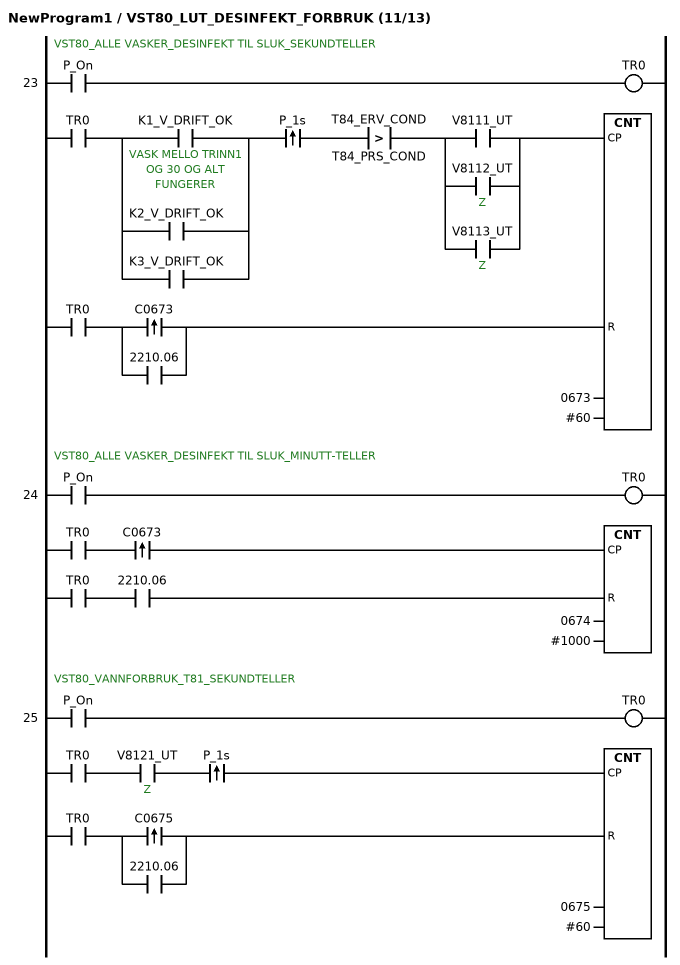
; [picture p24: NewProgram1 / VST80_LUT_DESINFEKT_FORBRUK, rungs 23-25]
; rung 23: VST80_ALLE VASKER_DESINFEKT TIL SLUK_SEKUNDTELLER
LD P_On
OUT TR0
LD K1_V_DRIFT_OK  ; VASK MELLO TRINN1 OG 30 OG ALT FUNGERER
OR K2_V_DRIFT_OK
OR K3_V_DRIFT_OK
ANDLD
@AND P_1s
AND>(320) T84_ERV_COND T84_PRS_COND
LD V8111_UT
OR V8112_UT  ; Z
OR V8113_UT  ; Z
ANDLD
LD TR0
@LD C0673
OR 2210.06
ANDLD
CNT 0673 #60
; rung 24: VST80_ALLE VASKER_DESINFEKT TIL SLUK_MINUTT-TELLER
LD P_On
OUT TR0
@AND C0673
LD TR0
AND 2210.06
CNT 0674 #1000
; rung 25: VST80_VANNFORBRUK_T81_SEKUNDTELLER
LD P_On
OUT TR0
AND V8121_UT  ; Z
@AND P_1s
LD TR0
@LD C0675
OR 2210.06
ANDLD
CNT 0675 #60

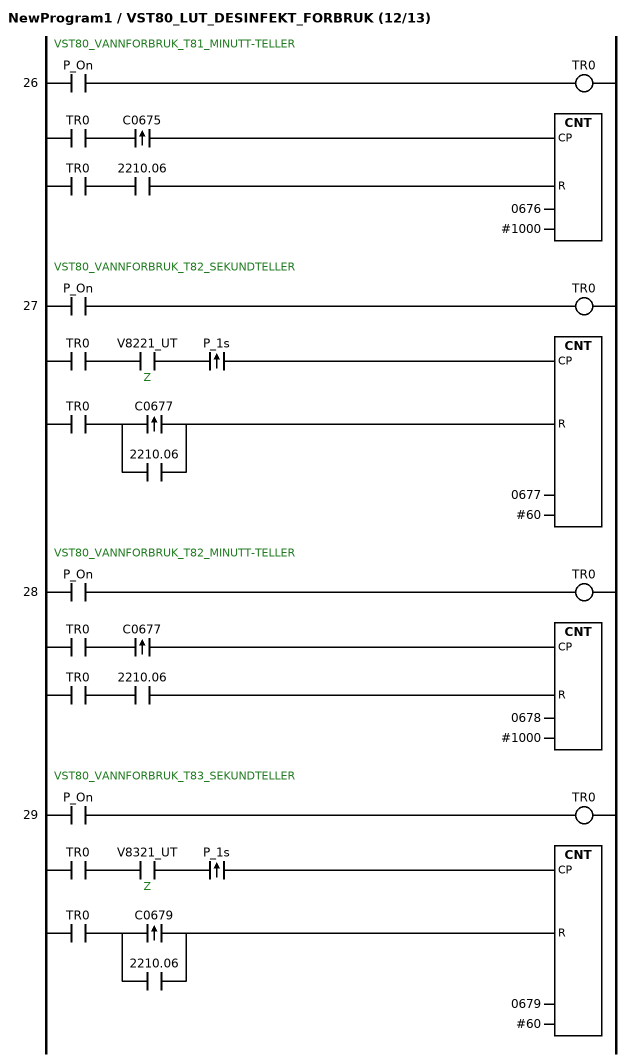
; rung 26: VST80_VANNFORBRUK_T81_MINUTT-TELLER
LD P_On
OUT TR0
@AND C0675
LD TR0
AND 2210.06
CNT 0676 #1000
; rung 27: VST80_VANNFORBRUK_T82_SEKUNDTELLER
LD P_On
OUT TR0
AND V8221_UT  ; Z
@AND P_1s
LD TR0
@LD C0677
OR 2210.06
ANDLD
CNT 0677 #60
; rung 28: VST80_VANNFORBRUK_T82_MINUTT-TELLER
LD P_On
OUT TR0
@AND C0677
LD TR0
AND 2210.06
CNT 0678 #1000
; rung 29: VST80_VANNFORBRUK_T83_SEKUNDTELLER
LD P_On
OUT TR0
AND V8321_UT  ; Z
@AND P_1s
LD TR0
@LD C0679
OR 2210.06
ANDLD
CNT 0679 #60

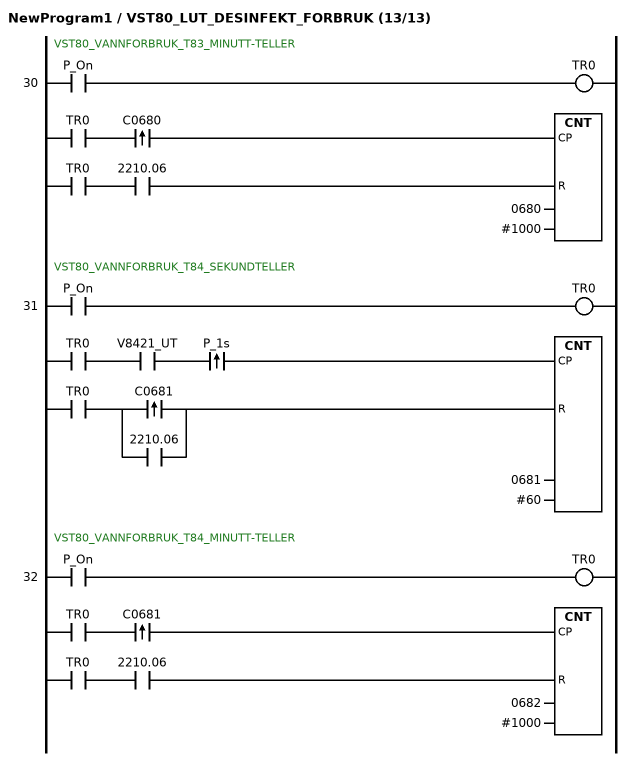
; rung 30: VST80_VANNFORBRUK_T83_MINUTT-TELLER
LD P_On
OUT TR0
@AND C0680
LD TR0
AND 2210.06
CNT 0680 #1000
; rung 31: VST80_VANNFORBRUK_T84_SEKUNDTELLER
LD P_On
OUT TR0
AND V8421_UT
@AND P_1s
LD TR0
@LD C0681
OR 2210.06
ANDLD
CNT 0681 #60
; rung 32: VST80_VANNFORBRUK_T84_MINUTT-TELLER
LD P_On
OUT TR0
@AND C0681
LD TR0
AND 2210.06
CNT 0682 #1000
; rung 33: Ingen_kommentar_funnet

### Section T81_NIVÅ

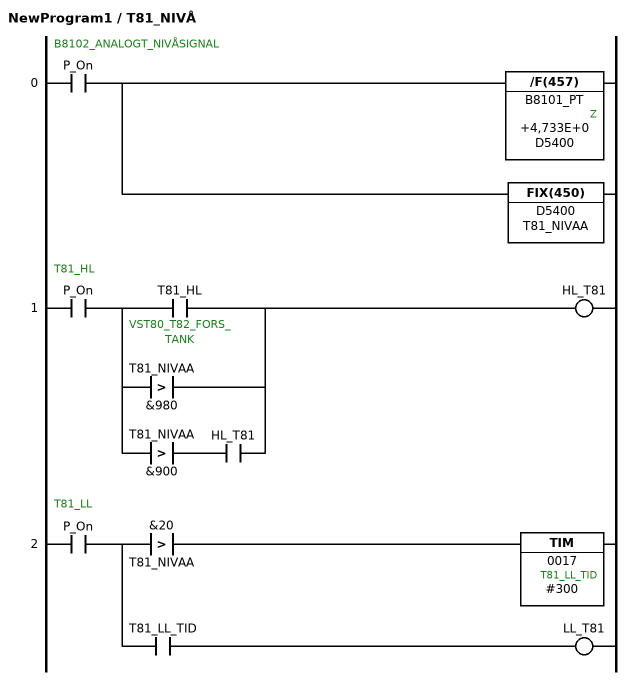
; rung 0: B8102_ANALOGT_NIVÅSIGNAL
LD P_On
/F(457) B8101_PT +4,733E+0 D5400  ; Z
FIX(450) D5400 T81_NIVAA
; rung 1: T81_HL
LD P_On
LD T81_HL  ; VST80_T82_FORS_TANK
OR>(320) T81_NIVAA &980
LD>(320) T81_NIVAA &900
AND HL_T81
ORLD
ANDLD
OUT HL_T81
; rung 2: T81_LL
LD P_On
OUT TR0
AND>(320) &20 T81_NIVAA
TIM 0017 #300  ; T81_LL_TID
LD TR0
AND T81_LL_TID
OUT LL_T81
; rung 3: Ingen_kommentar_funnet

### Section T81_FUNKSJONER_OBJEKTER
; Dette programmet styrer kommandoene til vaskestasjonen.

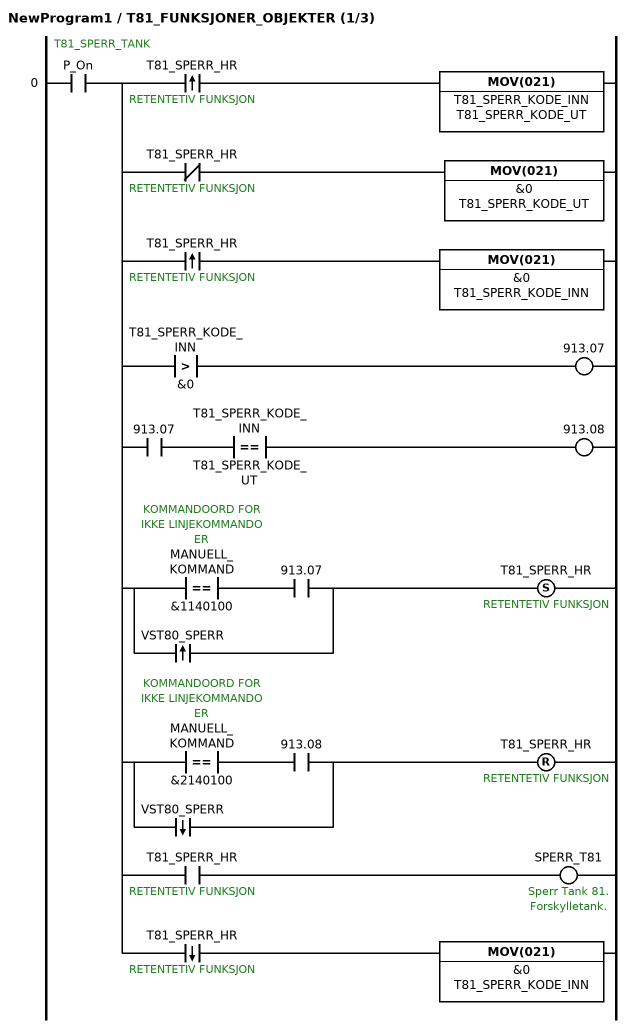
; rung 0: T81_SPERR_TANK
LD P_On
OUT TR0
@AND T81_SPERR_HR  ; RETENTETIV FUNKSJON
MOV(021) T81_SPERR_KODE_INN T81_SPERR_KODE_UT
LD TR0
ANDNOT T81_SPERR_HR  ; RETENTETIV FUNKSJON
MOV(021) &0 T81_SPERR_KODE_UT
LD TR0
@AND T81_SPERR_HR  ; RETENTETIV FUNKSJON
MOV(021) &0 T81_SPERR_KODE_INN
LD TR0
AND>(320) T81_SPERR_KODE_INN &0
OUT 913.07
LD TR0
AND 913.07
AND=(300) T81_SPERR_KODE_INN T81_SPERR_KODE_UT
OUT 913.08
LD TR0
LD=L(301) MANUELL_KOMMAND &1140100  ; KOMMANDOORD FOR IKKE LINJEKOMMANDOER
AND 913.07
@OR VST80_SPERR
ANDLD
SET T81_SPERR_HR  ; RETENTETIV FUNKSJON
LD TR0
LD=L(301) MANUELL_KOMMAND &2140100  ; KOMMANDOORD FOR IKKE LINJEKOMMANDOER
AND 913.08
%OR VST80_SPERR
ANDLD
RSET T81_SPERR_HR  ; RETENTETIV FUNKSJON
LD TR0
AND T81_SPERR_HR  ; RETENTETIV FUNKSJON
OUT SPERR_T81  ; Sperr Tank 81. Forskylletank.
LD TR0
%AND T81_SPERR_HR  ; RETENTETIV FUNKSJON
MOV(021) &0 T81_SPERR_KODE_INN

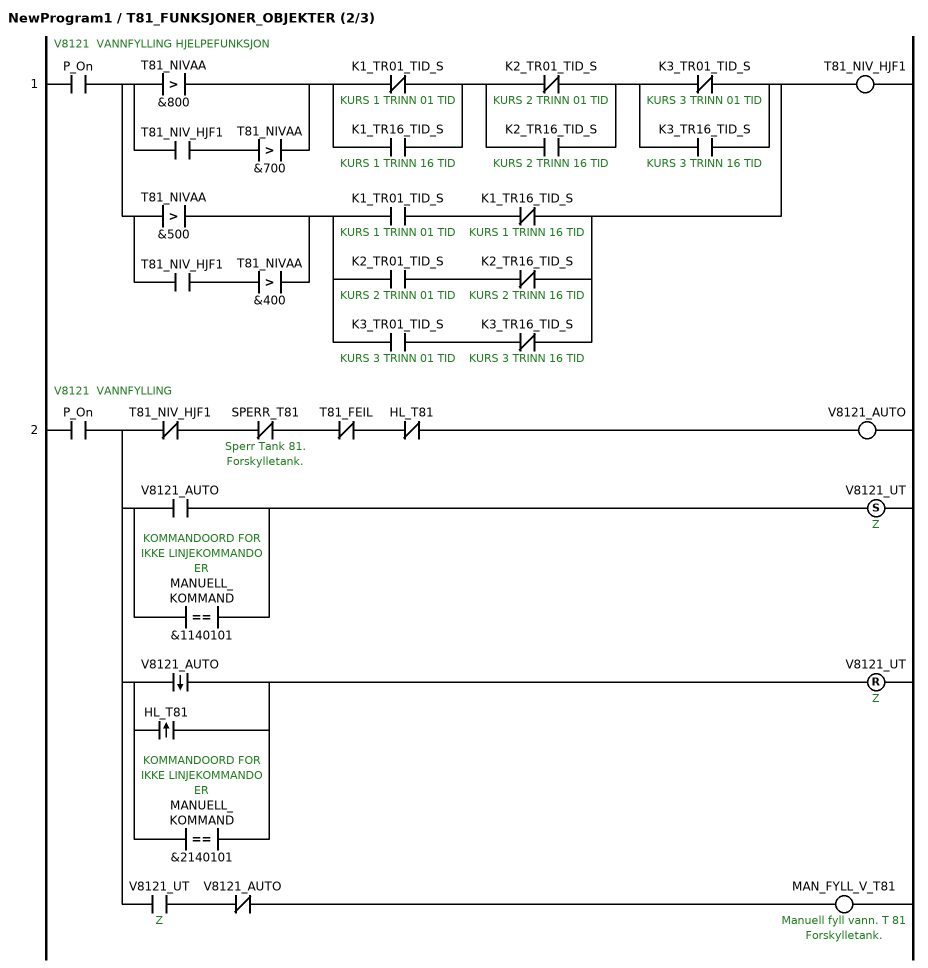
; rung 1: V8121  VANNFYLLING HJELPEFUNKSJON
LD P_On
LD>(320) T81_NIVAA &800
LD T81_NIV_HJF1
AND>(320) T81_NIVAA &700
ORLD
LDNOT K1_TR01_TID_S  ; KURS 1 TRINN 01 TID
OR K1_TR16_TID_S  ; KURS 1 TRINN 16 TID
ANDLD
LDNOT K2_TR01_TID_S  ; KURS 2 TRINN 01 TID
OR K2_TR16_TID_S  ; KURS 2 TRINN 16 TID
ANDLD
LDNOT K3_TR01_TID_S  ; KURS 3 TRINN 01 TID
OR K3_TR16_TID_S  ; KURS 3 TRINN 16 TID
ANDLD
LD>(320) T81_NIVAA &500
LD T81_NIV_HJF1
AND>(320) T81_NIVAA &400
ORLD
LD K1_TR01_TID_S  ; KURS 1 TRINN 01 TID
ANDNOT K1_TR16_TID_S  ; KURS 1 TRINN 16 TID
LD K2_TR01_TID_S  ; KURS 2 TRINN 01 TID
ANDNOT K2_TR16_TID_S  ; KURS 2 TRINN 16 TID
ORLD
LD K3_TR01_TID_S  ; KURS 3 TRINN 01 TID
ANDNOT K3_TR16_TID_S  ; KURS 3 TRINN 16 TID
ORLD
ANDLD
ORLD
ANDLD
OUT T81_NIV_HJF1
; rung 2: V8121  VANNFYLLING
LD P_On
OUT TR0
ANDNOT T81_NIV_HJF1
ANDNOT SPERR_T81  ; Sperr Tank 81. Forskylletank.
ANDNOT T81_FEIL
ANDNOT HL_T81
OUT V8121_AUTO
LD TR0
LD V8121_AUTO
OR=L(301) MANUELL_KOMMAND &1140101  ; KOMMANDOORD FOR IKKE LINJEKOMMANDOER
ANDLD
SET V8121_UT  ; Z
LD TR0
%LD V8121_AUTO
@OR HL_T81
OR=L(301) MANUELL_KOMMAND &2140101  ; KOMMANDOORD FOR IKKE LINJEKOMMANDOER
ANDLD
RSET V8121_UT  ; Z
LD TR0
AND V8121_UT  ; Z
ANDNOT V8121_AUTO
OUT MAN_FYLL_V_T81  ; Manuell fyll vann. T 81 Forskylletank.

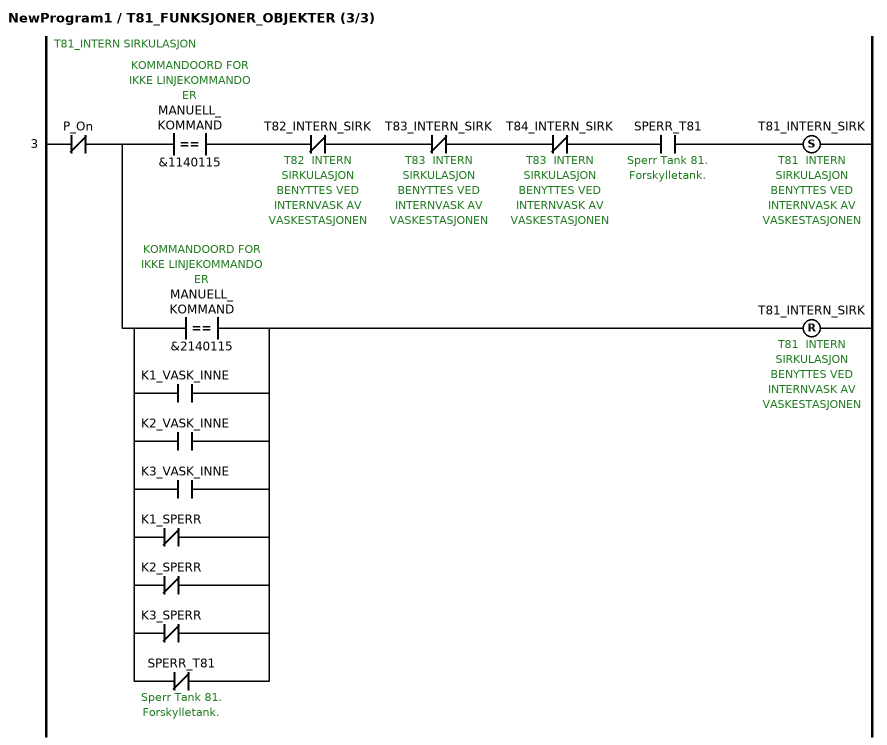
; rung 3: T81_INTERN SIRKULASJON
LDNOT P_On
OUT TR0
AND=L(301) MANUELL_KOMMAND &1140115  ; KOMMANDOORD FOR IKKE LINJEKOMMANDOER
ANDNOT T82_INTERN_SIRK  ; T82  INTERN SIRKULASJON BENYTTES VED INTERNVASK AV VASKESTASJONEN
ANDNOT T83_INTERN_SIRK  ; T83  INTERN SIRKULASJON BENYTTES VED INTERNVASK AV VASKESTASJONEN
ANDNOT T84_INTERN_SIRK  ; T83  INTERN SIRKULASJON BENYTTES VED INTERNVASK AV VASKESTASJONEN
AND SPERR_T81  ; Sperr Tank 81. Forskylletank.
SET T81_INTERN_SIRK  ; T81  INTERN SIRKULASJON BENYTTES VED INTERNVASK AV VASKESTASJONEN
LD TR0
LD=L(301) MANUELL_KOMMAND &2140115  ; KOMMANDOORD FOR IKKE LINJEKOMMANDOER
OR K1_VASK_INNE
OR K2_VASK_INNE
OR K3_VASK_INNE
ORNOT K1_SPERR
ORNOT K2_SPERR
ORNOT K3_SPERR
ORNOT SPERR_T81  ; Sperr Tank 81. Forskylletank.
ANDLD
RSET T81_INTERN_SIRK  ; T81  INTERN SIRKULASJON BENYTTES VED INTERNVASK AV VASKESTASJONEN
; rung 4: Ingen_kommentar_funnet

### Section T82_NIVÅ_TEMP_CONDUKTIVITET

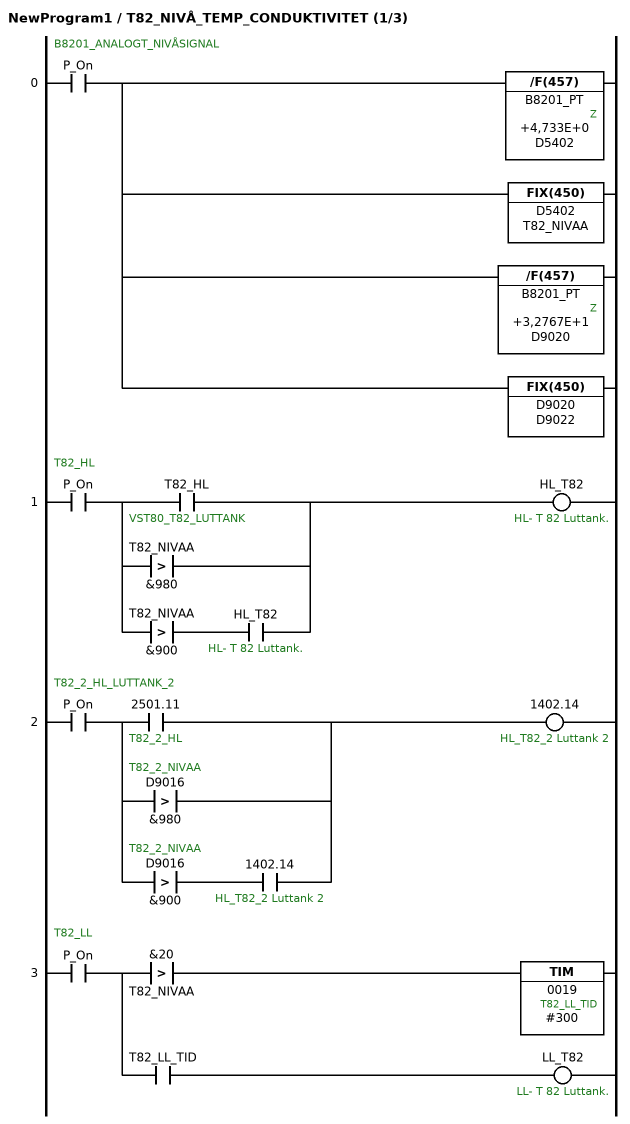
; rung 0: B8201_ANALOGT_NIVÅSIGNAL
LD P_On
/F(457) B8201_PT +4,733E+0 D5402  ; Z
FIX(450) D5402 T82_NIVAA
/F(457) B8201_PT +3,2767E+1 D9020  ; Z
FIX(450) D9020 D9022
; rung 1: T82_HL
LD P_On
LD T82_HL  ; VST80_T82_LUTTANK
OR>(320) T82_NIVAA &980
LD>(320) T82_NIVAA &900
AND HL_T82  ; HL- T 82 Luttank.
ORLD
ANDLD
OUT HL_T82  ; HL- T 82 Luttank.
; rung 2: T82_2_HL_LUTTANK_2
LD P_On
LD 2501.11  ; T82_2_HL
OR>(320) D9016 &980  ; T82_2_NIVAA
LD>(320) D9016 &900  ; T82_2_NIVAA
AND 1402.14  ; HL_T82_2 Luttank 2
ORLD
ANDLD
OUT 1402.14  ; HL_T82_2 Luttank 2
; rung 3: T82_LL
LD P_On
OUT TR0
AND>(320) &20 T82_NIVAA
TIM 0019 #300  ; T82_LL_TID
LD TR0
AND T82_LL_TID
OUT LL_T82  ; LL- T 82 Luttank.

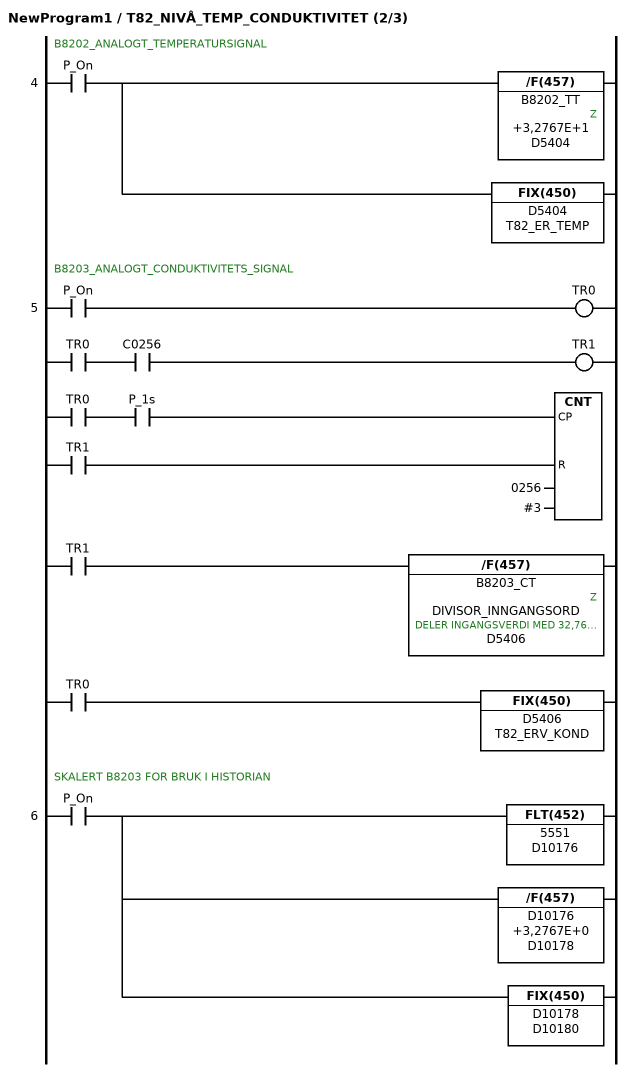
; rung 4: B8202_ANALOGT_TEMPERATURSIGNAL
LD P_On
/F(457) B8202_TT +3,2767E+1 D5404  ; Z
FIX(450) D5404 T82_ER_TEMP
; rung 5: B8203_ANALOGT_CONDUKTIVITETS_SIGNAL
LD P_On
OUT TR0
AND P_1s
LD TR0
AND C0256
OUT TR1
CNT 0256 #3
LD TR1
/F(457) B8203_CT DIVISOR_INNGANGSORD D5406  ; Z, DELER INGANGSVERDI MED 32,760 FOR OMREGNING TIL 0-1000
LD TR0
FIX(450) D5406 T82_ERV_KOND
; rung 6: SKALERT B8203 FOR BRUK I HISTORIAN
LD P_On
FLT(452) 5551 D10176
/F(457) D10176 +3,2767E+0 D10178
FIX(450) D10178 D10180

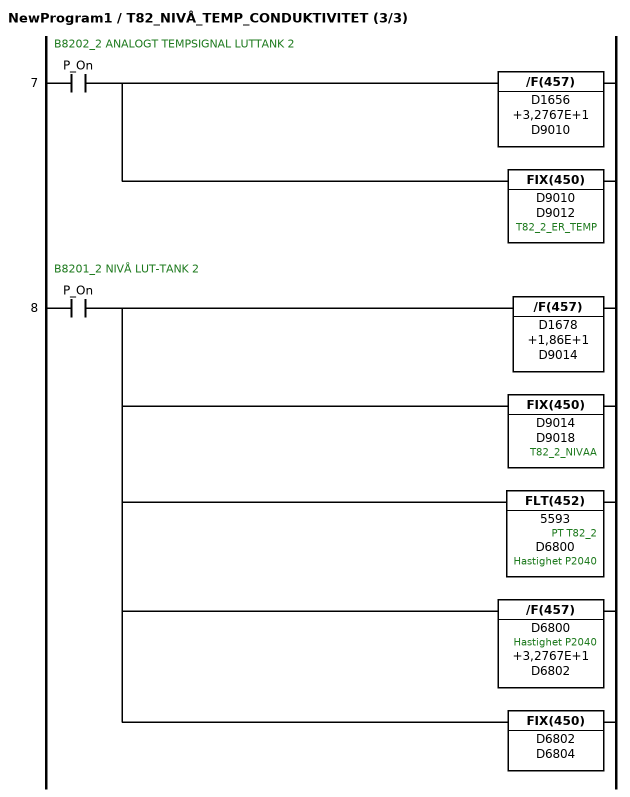
; rung 7: B8202_2 ANALOGT TEMPSIGNAL LUTTANK 2
LD P_On
/F(457) D1656 +3,2767E+1 D9010
FIX(450) D9010 D9012  ; T82_2_ER_TEMP
; rung 8: B8201_2 NIVÅ LUT-TANK 2
LD P_On
/F(457) D1678 +1,86E+1 D9014
FIX(450) D9014 D9018  ; T82_2_NIVAA
FLT(452) 5593 D6800  ; PT T82_2, Hastighet P2040
/F(457) D6800 +3,2767E+1 D6802  ; Hastighet P2040
FIX(450) D6802 D6804
; rung 9: Ingen_kommentar_funnet

### Section T82_FUNKSJONER_OBJEKTER

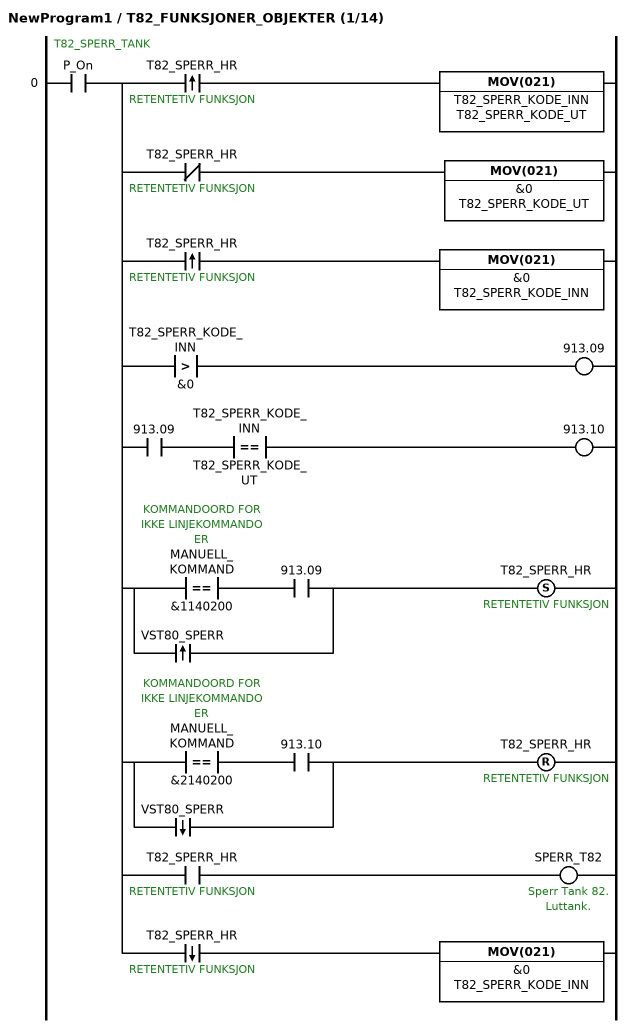
; rung 0: T82_SPERR_TANK
LD P_On
OUT TR0
@AND T82_SPERR_HR  ; RETENTETIV FUNKSJON
MOV(021) T82_SPERR_KODE_INN T82_SPERR_KODE_UT
LD TR0
ANDNOT T82_SPERR_HR  ; RETENTETIV FUNKSJON
MOV(021) &0 T82_SPERR_KODE_UT
LD TR0
@AND T82_SPERR_HR  ; RETENTETIV FUNKSJON
MOV(021) &0 T82_SPERR_KODE_INN
LD TR0
AND>(320) T82_SPERR_KODE_INN &0
OUT 913.09
LD TR0
AND 913.09
AND=(300) T82_SPERR_KODE_INN T82_SPERR_KODE_UT
OUT 913.10
LD TR0
LD=L(301) MANUELL_KOMMAND &1140200  ; KOMMANDOORD FOR IKKE LINJEKOMMANDOER
AND 913.09
@OR VST80_SPERR
ANDLD
SET T82_SPERR_HR  ; RETENTETIV FUNKSJON
LD TR0
LD=L(301) MANUELL_KOMMAND &2140200  ; KOMMANDOORD FOR IKKE LINJEKOMMANDOER
AND 913.10
%OR VST80_SPERR
ANDLD
RSET T82_SPERR_HR  ; RETENTETIV FUNKSJON
LD TR0
AND T82_SPERR_HR  ; RETENTETIV FUNKSJON
OUT SPERR_T82  ; Sperr Tank 82. Luttank.
LD TR0
%AND T82_SPERR_HR  ; RETENTETIV FUNKSJON
MOV(021) &0 T82_SPERR_KODE_INN

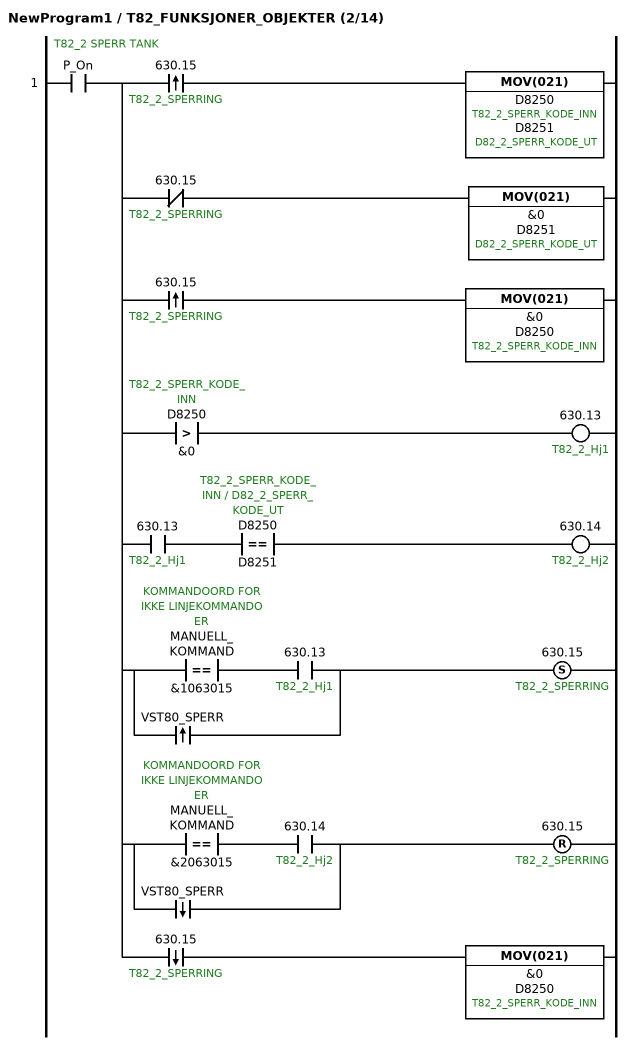
; rung 1: T82_2 SPERR TANK
LD P_On
OUT TR0
@AND 630.15  ; T82_2_SPERRING
MOV(021) D8250 D8251  ; T82_2_SPERR_KODE_INN, D82_2_SPERR_KODE_UT
LD TR0
ANDNOT 630.15  ; T82_2_SPERRING
MOV(021) &0 D8251  ; D82_2_SPERR_KODE_UT
LD TR0
@AND 630.15  ; T82_2_SPERRING
MOV(021) &0 D8250  ; T82_2_SPERR_KODE_INN
LD TR0
AND>(320) D8250 &0  ; T82_2_SPERR_KODE_INN
OUT 630.13  ; T82_2_Hj1
LD TR0
AND 630.13  ; T82_2_Hj1
AND=(300) D8250 D8251  ; T82_2_SPERR_KODE_INN, D82_2_SPERR_KODE_UT
OUT 630.14  ; T82_2_Hj2
LD TR0
LD=L(301) MANUELL_KOMMAND &1063015  ; KOMMANDOORD FOR IKKE LINJEKOMMANDOER
AND 630.13  ; T82_2_Hj1
@OR VST80_SPERR
ANDLD
SET 630.15  ; T82_2_SPERRING
LD TR0
LD=L(301) MANUELL_KOMMAND &2063015  ; KOMMANDOORD FOR IKKE LINJEKOMMANDOER
AND 630.14  ; T82_2_Hj2
%OR VST80_SPERR
ANDLD
RSET 630.15  ; T82_2_SPERRING
LD TR0
%AND 630.15  ; T82_2_SPERRING
MOV(021) &0 D8250  ; T82_2_SPERR_KODE_INN
; rung 2: SIGNALER DRIFT PASTEURVASK FELLES FOR FYLLING AV TANK 82_83

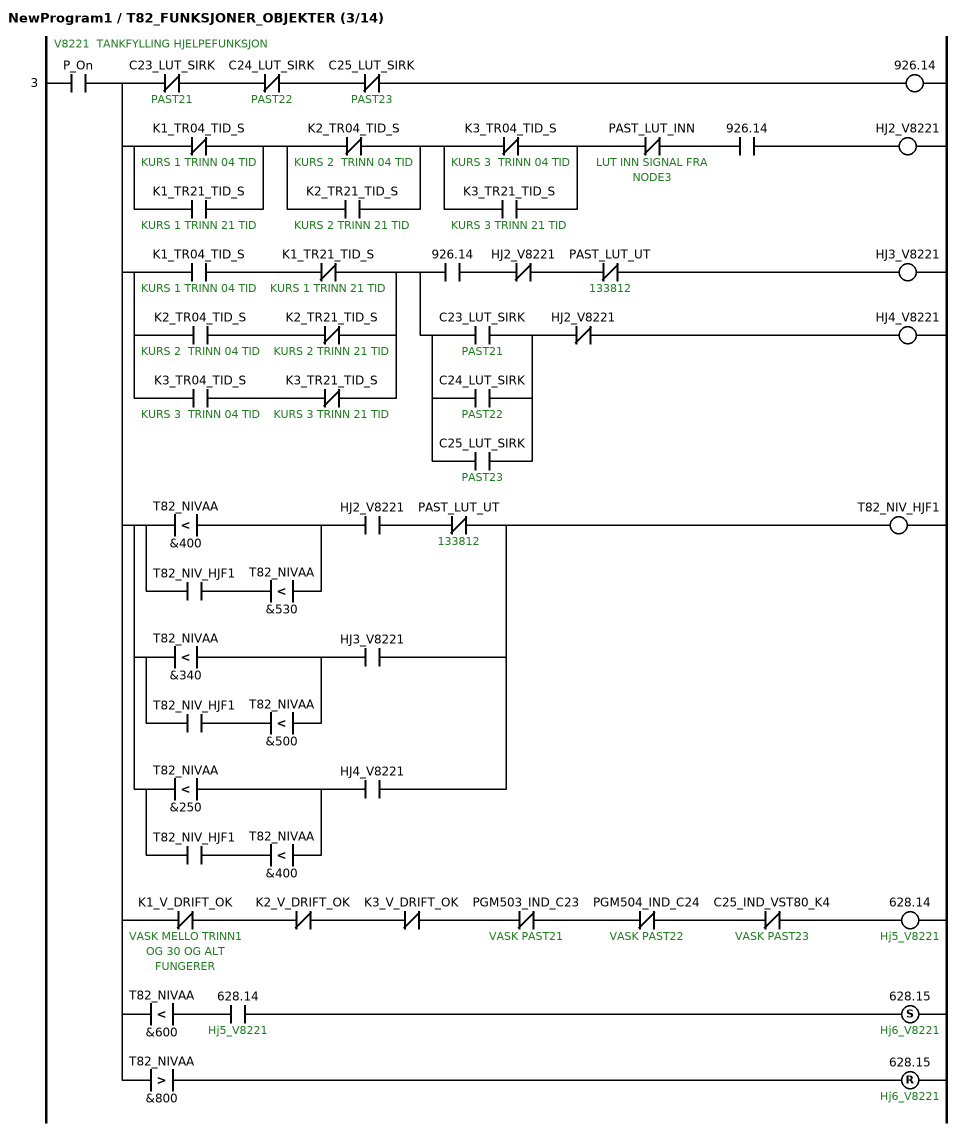
; rung 3: V8221  TANKFYLLING HJELPEFUNKSJON
LD P_On
OUT TR0
ANDNOT C23_LUT_SIRK  ; PAST21
ANDNOT C24_LUT_SIRK  ; PAST22
ANDNOT C25_LUT_SIRK  ; PAST23
OUT 926.14
LD TR0
LDNOT K1_TR04_TID_S  ; KURS 1 TRINN 04 TID
OR K1_TR21_TID_S  ; KURS 1 TRINN 21 TID
ANDLD
LDNOT K2_TR04_TID_S  ; KURS 2  TRINN 04 TID
OR K2_TR21_TID_S  ; KURS 2 TRINN 21 TID
ANDLD
LDNOT K3_TR04_TID_S  ; KURS 3  TRINN 04 TID
OR K3_TR21_TID_S  ; KURS 3 TRINN 21 TID
ANDLD
ANDNOT PAST_LUT_INN  ; LUT INN SIGNAL FRA NODE3
AND 926.14
OUT HJ2_V8221
LD TR0
LD K1_TR04_TID_S  ; KURS 1 TRINN 04 TID
ANDNOT K1_TR21_TID_S  ; KURS 1 TRINN 21 TID
LD K2_TR04_TID_S  ; KURS 2  TRINN 04 TID
ANDNOT K2_TR21_TID_S  ; KURS 2 TRINN 21 TID
ORLD
LD K3_TR04_TID_S  ; KURS 3  TRINN 04 TID
ANDNOT K3_TR21_TID_S  ; KURS 3 TRINN 21 TID
ORLD
ANDLD
OUT TR1
AND 926.14
ANDNOT HJ2_V8221
ANDNOT PAST_LUT_UT  ; 133812
OUT HJ3_V8221
LD TR1
LD C23_LUT_SIRK  ; PAST21
OR C24_LUT_SIRK  ; PAST22
OR C25_LUT_SIRK  ; PAST23
ANDLD
ANDNOT HJ2_V8221
OUT HJ4_V8221
LD TR0
LD<(310) T82_NIVAA &400
LD T82_NIV_HJF1
AND<(310) T82_NIVAA &530
ORLD
AND HJ2_V8221
ANDNOT PAST_LUT_UT  ; 133812
LD<(310) T82_NIVAA &340
LD T82_NIV_HJF1
AND<(310) T82_NIVAA &500
ORLD
AND HJ3_V8221
ORLD
LD<(310) T82_NIVAA &250
LD T82_NIV_HJF1
AND<(310) T82_NIVAA &400
ORLD
AND HJ4_V8221
ORLD
ANDLD
OUT T82_NIV_HJF1
LD TR0
ANDNOT K1_V_DRIFT_OK  ; VASK MELLO TRINN1 OG 30 OG ALT FUNGERER
ANDNOT K2_V_DRIFT_OK
ANDNOT K3_V_DRIFT_OK
ANDNOT PGM503_IND_C23  ; VASK PAST21
ANDNOT PGM504_IND_C24  ; VASK PAST22
ANDNOT C25_IND_VST80_K4  ; VASK PAST23
OUT 628.14  ; Hj5_V8221
LD TR0
AND<(310) T82_NIVAA &600
AND 628.14  ; Hj5_V8221
SET 628.15  ; Hj6_V8221
LD TR0
AND>(320) T82_NIVAA &800
RSET 628.15  ; Hj6_V8221

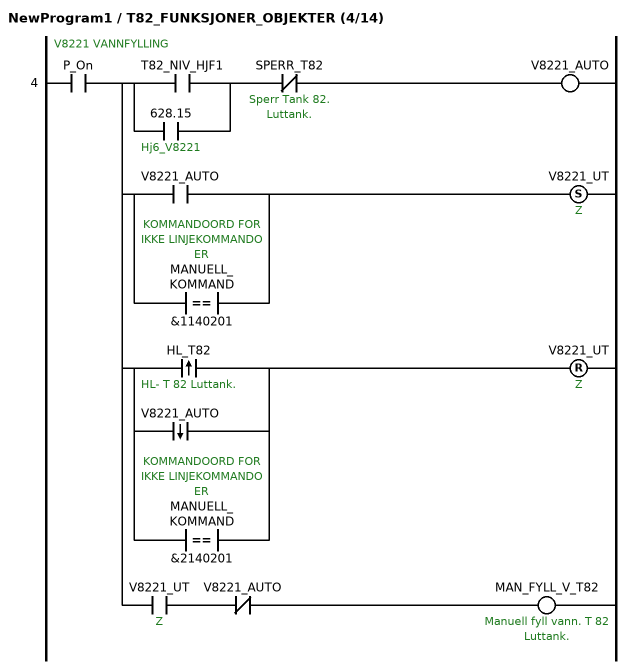
; rung 4: V8221 VANNFYLLING
LD P_On
OUT TR0
LD T82_NIV_HJF1
OR 628.15  ; Hj6_V8221
ANDLD
ANDNOT SPERR_T82  ; Sperr Tank 82. Luttank.
OUT V8221_AUTO
LD TR0
LD V8221_AUTO
OR=L(301) MANUELL_KOMMAND &1140201  ; KOMMANDOORD FOR IKKE LINJEKOMMANDOER
ANDLD
SET V8221_UT  ; Z
LD TR0
@LD HL_T82  ; HL- T 82 Luttank.
%OR V8221_AUTO
OR=L(301) MANUELL_KOMMAND &2140201  ; KOMMANDOORD FOR IKKE LINJEKOMMANDOER
ANDLD
RSET V8221_UT  ; Z
LD TR0
AND V8221_UT  ; Z
ANDNOT V8221_AUTO
OUT MAN_FYLL_V_T82  ; Manuell fyll vann. T 82 Luttank.

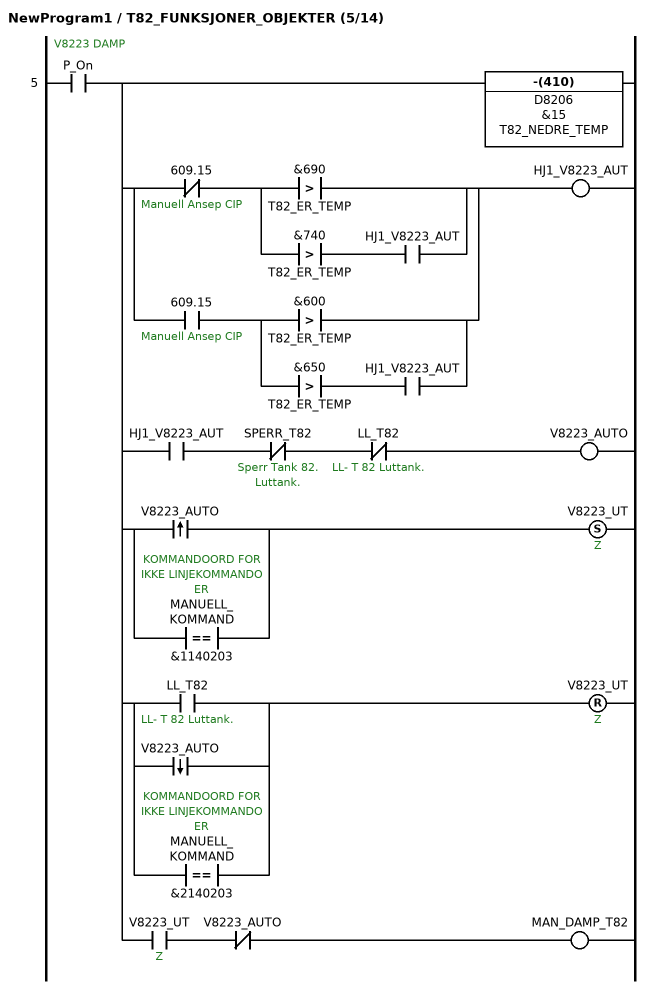
; rung 5: V8223 DAMP
LD P_On
OUT TR0
-(410) D8206 &15 T82_NEDRE_TEMP
LDNOT 609.15  ; Manuell Ansep CIP
LD>(320) &690 T82_ER_TEMP
LD>(320) &740 T82_ER_TEMP
AND HJ1_V8223_AUT
ORLD
ANDLD
LD 609.15  ; Manuell Ansep CIP
LD>(320) &600 T82_ER_TEMP
LD>(320) &650 T82_ER_TEMP
AND HJ1_V8223_AUT
ORLD
ANDLD
ORLD
ANDLD
OUT HJ1_V8223_AUT
LD TR0
AND HJ1_V8223_AUT
ANDNOT SPERR_T82  ; Sperr Tank 82. Luttank.
ANDNOT LL_T82  ; LL- T 82 Luttank.
OUT V8223_AUTO
LD TR0
@LD V8223_AUTO
OR=L(301) MANUELL_KOMMAND &1140203  ; KOMMANDOORD FOR IKKE LINJEKOMMANDOER
ANDLD
SET V8223_UT  ; Z
LD TR0
LD LL_T82  ; LL- T 82 Luttank.
%OR V8223_AUTO
OR=L(301) MANUELL_KOMMAND &2140203  ; KOMMANDOORD FOR IKKE LINJEKOMMANDOER
ANDLD
RSET V8223_UT  ; Z
LD TR0
AND V8223_UT  ; Z
ANDNOT V8223_AUTO
OUT MAN_DAMP_T82

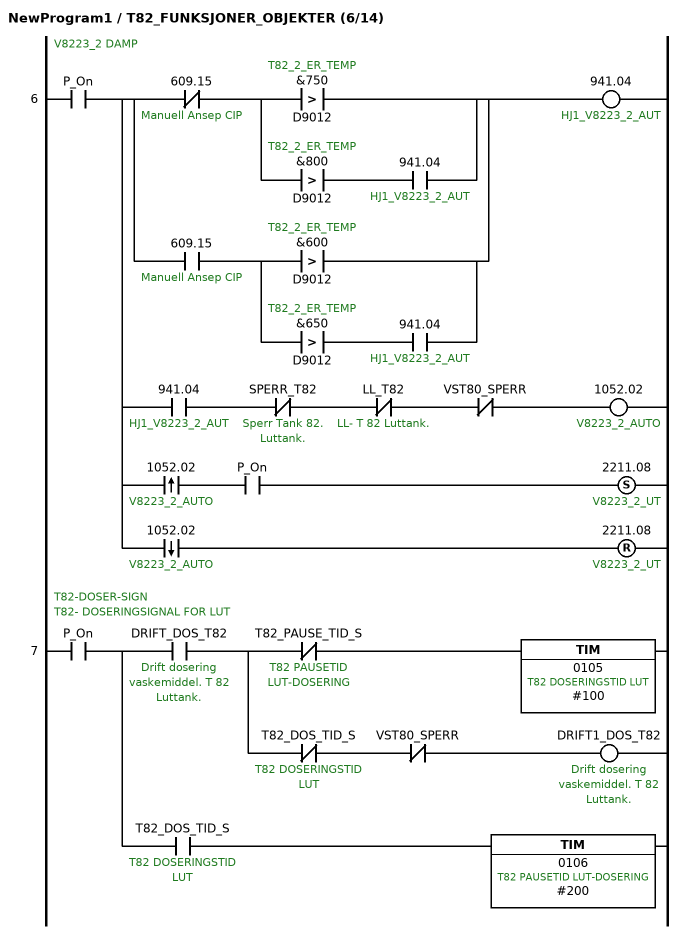
; rung 6: V8223_2 DAMP
LD P_On
OUT TR0
LDNOT 609.15  ; Manuell Ansep CIP
LD>(320) &750 D9012  ; T82_2_ER_TEMP
LD>(320) &800 D9012  ; T82_2_ER_TEMP
AND 941.04  ; HJ1_V8223_2_AUT
ORLD
ANDLD
LD 609.15  ; Manuell Ansep CIP
LD>(320) &600 D9012  ; T82_2_ER_TEMP
LD>(320) &650 D9012  ; T82_2_ER_TEMP
AND 941.04  ; HJ1_V8223_2_AUT
ORLD
ANDLD
ORLD
ANDLD
OUT 941.04  ; HJ1_V8223_2_AUT
LD TR0
AND 941.04  ; HJ1_V8223_2_AUT
ANDNOT SPERR_T82  ; Sperr Tank 82. Luttank.
ANDNOT LL_T82  ; LL- T 82 Luttank.
ANDNOT VST80_SPERR
OUT 1052.02  ; V8223_2_AUTO
LD TR0
@AND 1052.02  ; V8223_2_AUTO
AND P_On
SET 2211.08  ; V8223_2_UT
LD TR0
%AND 1052.02  ; V8223_2_AUTO
RSET 2211.08  ; V8223_2_UT
; rung 7: T82-DOSER-SIGN / T82- DOSERINGSIGNAL FOR LUT
LD P_On
OUT TR0
AND DRIFT_DOS_T82  ; Drift dosering vaskemiddel. T 82 Luttank.
OUT TR1
ANDNOT T82_PAUSE_TID_S  ; T82 PAUSETID LUT-DOSERING
TIM 0105 #100  ; T82 DOSERINGSTID LUT
LD TR1
ANDNOT T82_DOS_TID_S  ; T82 DOSERINGSTID LUT
ANDNOT VST80_SPERR
OUT DRIFT1_DOS_T82  ; Drift dosering vaskemiddel. T 82 Luttank.
LD TR0
AND T82_DOS_TID_S  ; T82 DOSERINGSTID LUT
TIM 0106 #200  ; T82 PAUSETID LUT-DOSERING

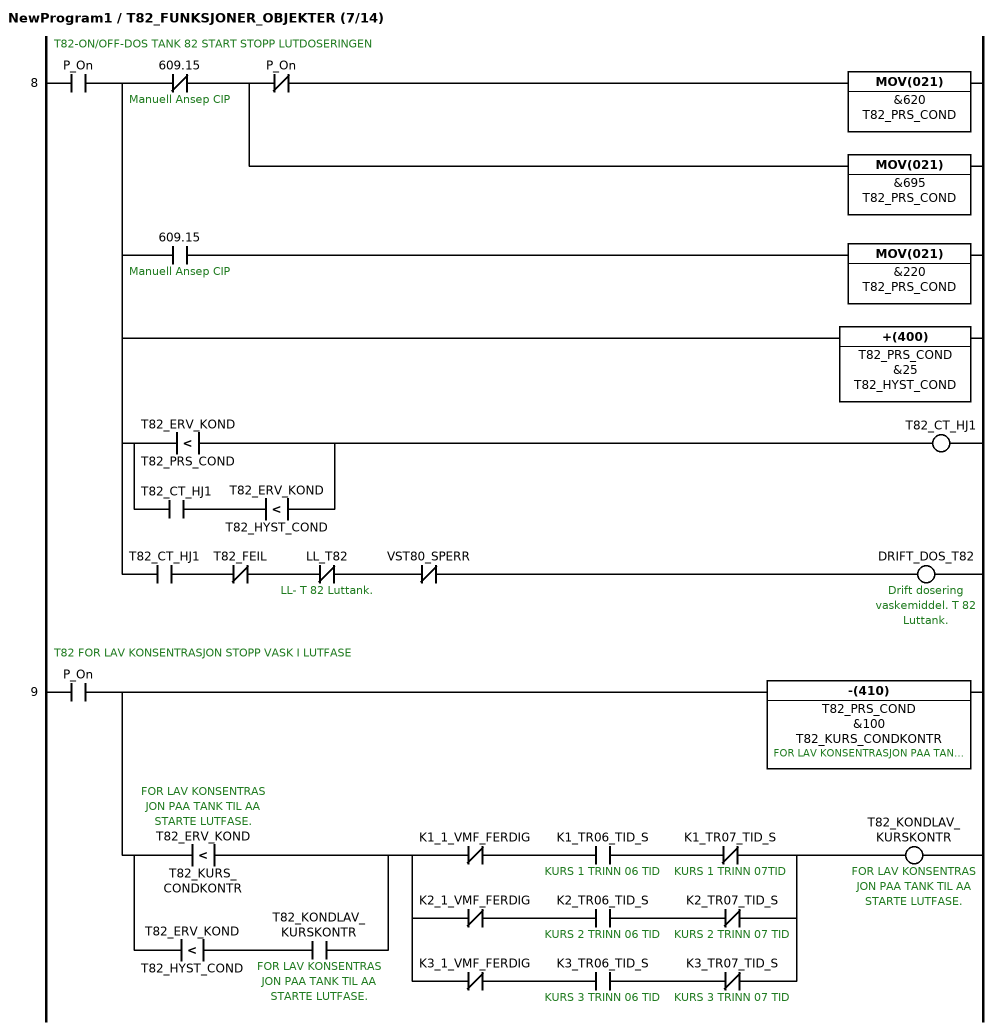
; rung 8: T82-ON/OFF-DOS TANK 82 START STOPP LUTDOSERINGEN
LD P_On
OUT TR0
ANDNOT 609.15  ; Manuell Ansep CIP
OUT TR1
ANDNOT P_On
MOV(021) &620 T82_PRS_COND
LD TR1
MOV(021) &695 T82_PRS_COND
LD TR0
AND 609.15  ; Manuell Ansep CIP
MOV(021) &220 T82_PRS_COND
LD TR0
+(400) T82_PRS_COND &25 T82_HYST_COND
LD<(310) T82_ERV_KOND T82_PRS_COND
LD T82_CT_HJ1
AND<(310) T82_ERV_KOND T82_HYST_COND
ORLD
ANDLD
OUT T82_CT_HJ1
LD TR0
AND T82_CT_HJ1
ANDNOT T82_FEIL
ANDNOT LL_T82  ; LL- T 82 Luttank.
ANDNOT VST80_SPERR
OUT DRIFT_DOS_T82  ; Drift dosering vaskemiddel. T 82 Luttank.
; rung 9: T82 FOR LAV KONSENTRASJON STOPP VASK I LUTFASE
LD P_On
-(410) T82_PRS_COND &100 T82_KURS_CONDKONTR  ; FOR LAV KONSENTRASJON PAA TANK TIL AA STARTE LUTFASE.
LD<(310) T82_ERV_KOND T82_KURS_CONDKONTR  ; FOR LAV KONSENTRASJON PAA TANK TIL AA STARTE LUTFASE.
LD<(310) T82_ERV_KOND T82_HYST_COND
AND T82_KONDLAV_KURSKONTR  ; FOR LAV KONSENTRASJON PAA TANK TIL AA STARTE LUTFASE.
ORLD
ANDLD
LDNOT K1_1_VMF_FERDIG
AND K1_TR06_TID_S  ; KURS 1 TRINN 06 TID
ANDNOT K1_TR07_TID_S  ; KURS 1 TRINN 07TID
LDNOT K2_1_VMF_FERDIG
AND K2_TR06_TID_S  ; KURS 2 TRINN 06 TID
ANDNOT K2_TR07_TID_S  ; KURS 2 TRINN 07 TID
ORLD
LDNOT K3_1_VMF_FERDIG
AND K3_TR06_TID_S  ; KURS 3 TRINN 06 TID
ANDNOT K3_TR07_TID_S  ; KURS 3 TRINN 07 TID
ORLD
ANDLD
OUT T82_KONDLAV_KURSKONTR  ; FOR LAV KONSENTRASJON PAA TANK TIL AA STARTE LUTFASE.

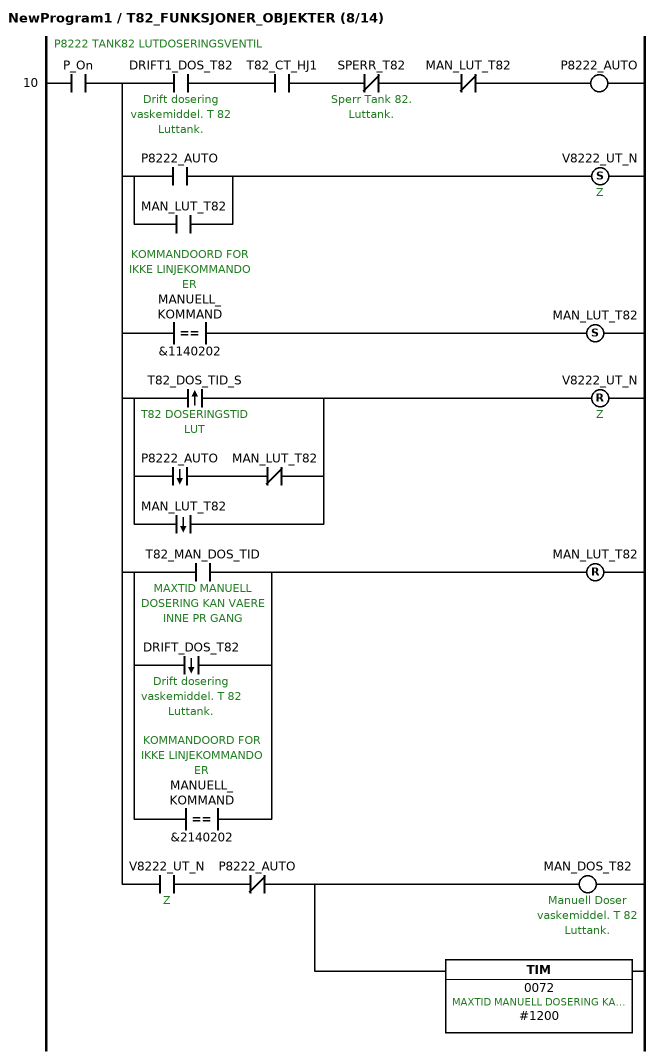
; rung 10: P8222 TANK82 LUTDOSERINGSVENTIL
LD P_On
OUT TR0
AND DRIFT1_DOS_T82  ; Drift dosering vaskemiddel. T 82 Luttank.
AND T82_CT_HJ1
ANDNOT SPERR_T82  ; Sperr Tank 82. Luttank.
ANDNOT MAN_LUT_T82
OUT P8222_AUTO
LD TR0
LD P8222_AUTO
OR MAN_LUT_T82
ANDLD
SET V8222_UT_N  ; Z
LD TR0
AND=L(301) MANUELL_KOMMAND &1140202  ; KOMMANDOORD FOR IKKE LINJEKOMMANDOER
SET MAN_LUT_T82
LD TR0
@LD T82_DOS_TID_S  ; T82 DOSERINGSTID LUT
%LD P8222_AUTO
ANDNOT MAN_LUT_T82
ORLD
%OR MAN_LUT_T82
ANDLD
RSET V8222_UT_N  ; Z
LD TR0
LD T82_MAN_DOS_TID  ; MAXTID MANUELL DOSERING KAN VAERE INNE PR GANG
%OR DRIFT_DOS_T82  ; Drift dosering vaskemiddel. T 82 Luttank.
OR=L(301) MANUELL_KOMMAND &2140202  ; KOMMANDOORD FOR IKKE LINJEKOMMANDOER
ANDLD
RSET MAN_LUT_T82
LD TR0
AND V8222_UT_N  ; Z
ANDNOT P8222_AUTO
OUT MAN_DOS_T82  ; Manuell Doser vaskemiddel. T 82 Luttank.
TIM 0072 #1200  ; MAXTID MANUELL DOSERING KAN VAERE INNE PR GANG

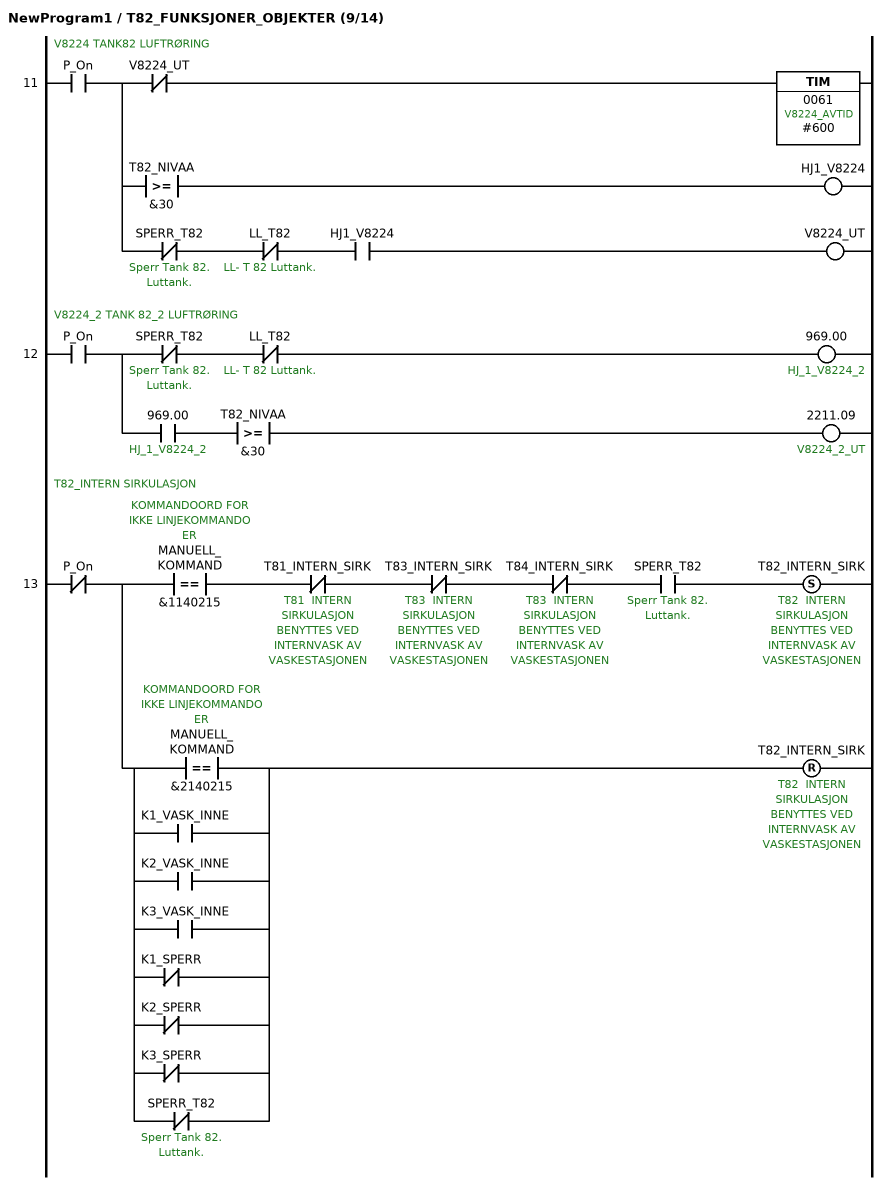
; rung 11: V8224 TANK82 LUFTRØRING
LD P_On
OUT TR0
ANDNOT V8224_UT
TIM 0061 #600  ; V8224_AVTID
LD TR0
AND>=(325) T82_NIVAA &30
OUT HJ1_V8224
LD TR0
ANDNOT SPERR_T82  ; Sperr Tank 82. Luttank.
ANDNOT LL_T82  ; LL- T 82 Luttank.
AND HJ1_V8224
OUT V8224_UT
; rung 12: V8224_2 TANK 82_2 LUFTRØRING
LD P_On
OUT TR0
ANDNOT SPERR_T82  ; Sperr Tank 82. Luttank.
ANDNOT LL_T82  ; LL- T 82 Luttank.
OUT 969.00  ; HJ_1_V8224_2
LD TR0
AND 969.00  ; HJ_1_V8224_2
AND>=(325) T82_NIVAA &30
OUT 2211.09  ; V8224_2_UT
; rung 13: T82_INTERN SIRKULASJON
LDNOT P_On
OUT TR0
AND=L(301) MANUELL_KOMMAND &1140215  ; KOMMANDOORD FOR IKKE LINJEKOMMANDOER
ANDNOT T81_INTERN_SIRK  ; T81  INTERN SIRKULASJON BENYTTES VED INTERNVASK AV VASKESTASJONEN
ANDNOT T83_INTERN_SIRK  ; T83  INTERN SIRKULASJON BENYTTES VED INTERNVASK AV VASKESTASJONEN
ANDNOT T84_INTERN_SIRK  ; T83  INTERN SIRKULASJON BENYTTES VED INTERNVASK AV VASKESTASJONEN
AND SPERR_T82  ; Sperr Tank 82. Luttank.
SET T82_INTERN_SIRK  ; T82  INTERN SIRKULASJON BENYTTES VED INTERNVASK AV VASKESTASJONEN
LD TR0
LD=L(301) MANUELL_KOMMAND &2140215  ; KOMMANDOORD FOR IKKE LINJEKOMMANDOER
OR K1_VASK_INNE
OR K2_VASK_INNE
OR K3_VASK_INNE
ORNOT K1_SPERR
ORNOT K2_SPERR
ORNOT K3_SPERR
ORNOT SPERR_T82  ; Sperr Tank 82. Luttank.
ANDLD
RSET T82_INTERN_SIRK  ; T82  INTERN SIRKULASJON BENYTTES VED INTERNVASK AV VASKESTASJONEN

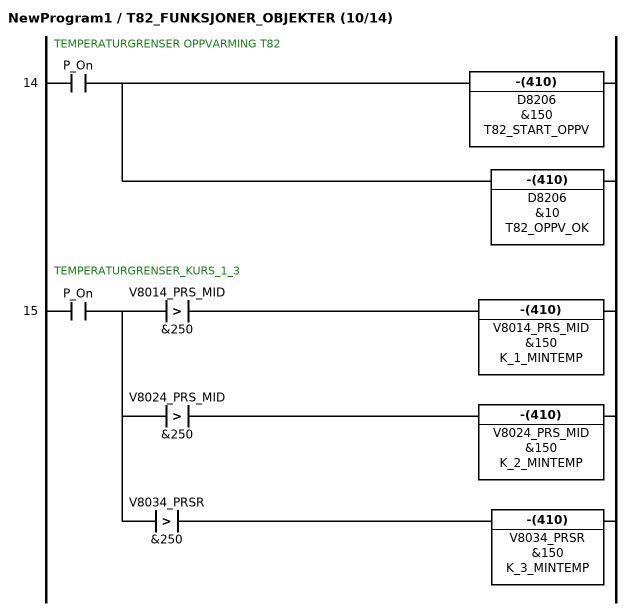
; rung 14: TEMPERATURGRENSER OPPVARMING T82
LD P_On
-(410) D8206 &150 T82_START_OPPV
-(410) D8206 &10 T82_OPPV_OK
; rung 15: TEMPERATURGRENSER_KURS_1_3
LD P_On
OUT TR0
AND>(320) V8014_PRS_MID &250
-(410) V8014_PRS_MID &150 K_1_MINTEMP
LD TR0
AND>(320) V8024_PRS_MID &250
-(410) V8024_PRS_MID &150 K_2_MINTEMP
LD TR0
AND>(320) V8034_PRSR &250
-(410) V8034_PRSR &150 K_3_MINTEMP

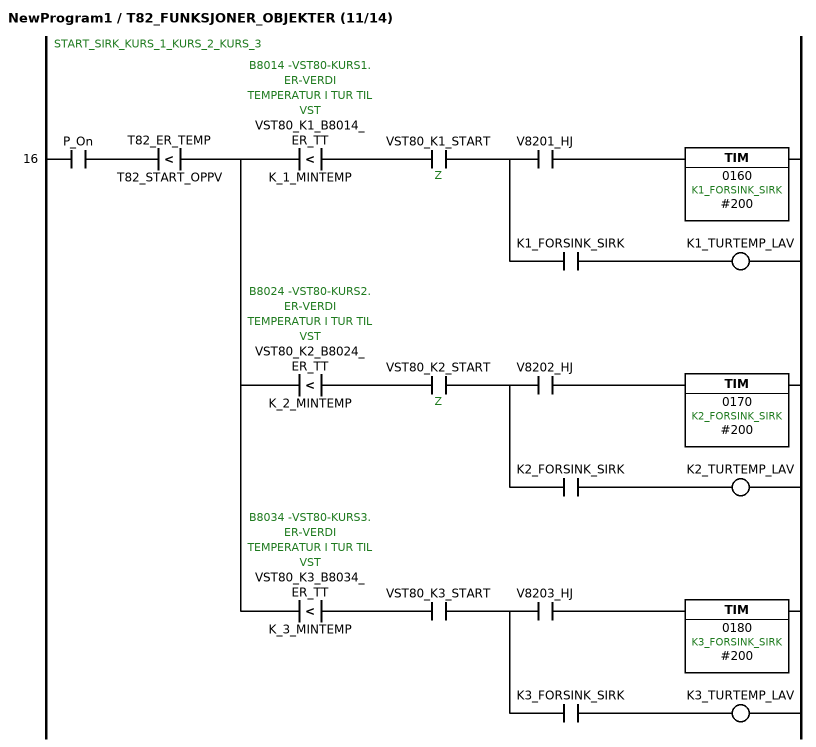
; rung 16: START_SIRK_KURS_1_KURS_2_KURS_3
LD P_On
AND<(310) T82_ER_TEMP T82_START_OPPV
OUT TR0
AND<(310) VST80_K1_B8014_ER_TT K_1_MINTEMP  ; B8014 -VST80-KURS1. ER-VERDI TEMPERATUR I TUR TIL VST
AND VST80_K1_START  ; Z
OUT TR1
AND V8201_HJ
TIM 0160 #200  ; K1_FORSINK_SIRK
LD TR1
AND K1_FORSINK_SIRK
OUT K1_TURTEMP_LAV
LD TR0
AND<(310) VST80_K2_B8024_ER_TT K_2_MINTEMP  ; B8024 -VST80-KURS2. ER-VERDI TEMPERATUR I TUR TIL VST
AND VST80_K2_START  ; Z
OUT TR1
AND V8202_HJ
TIM 0170 #200  ; K2_FORSINK_SIRK
LD TR1
AND K2_FORSINK_SIRK
OUT K2_TURTEMP_LAV
LD TR0
AND<(310) VST80_K3_B8034_ER_TT K_3_MINTEMP  ; B8034 -VST80-KURS3. ER-VERDI TEMPERATUR I TUR TIL VST
AND VST80_K3_START
OUT TR0
AND V8203_HJ
TIM 0180 #200  ; K3_FORSINK_SIRK
LD TR0
AND K3_FORSINK_SIRK
OUT K3_TURTEMP_LAV

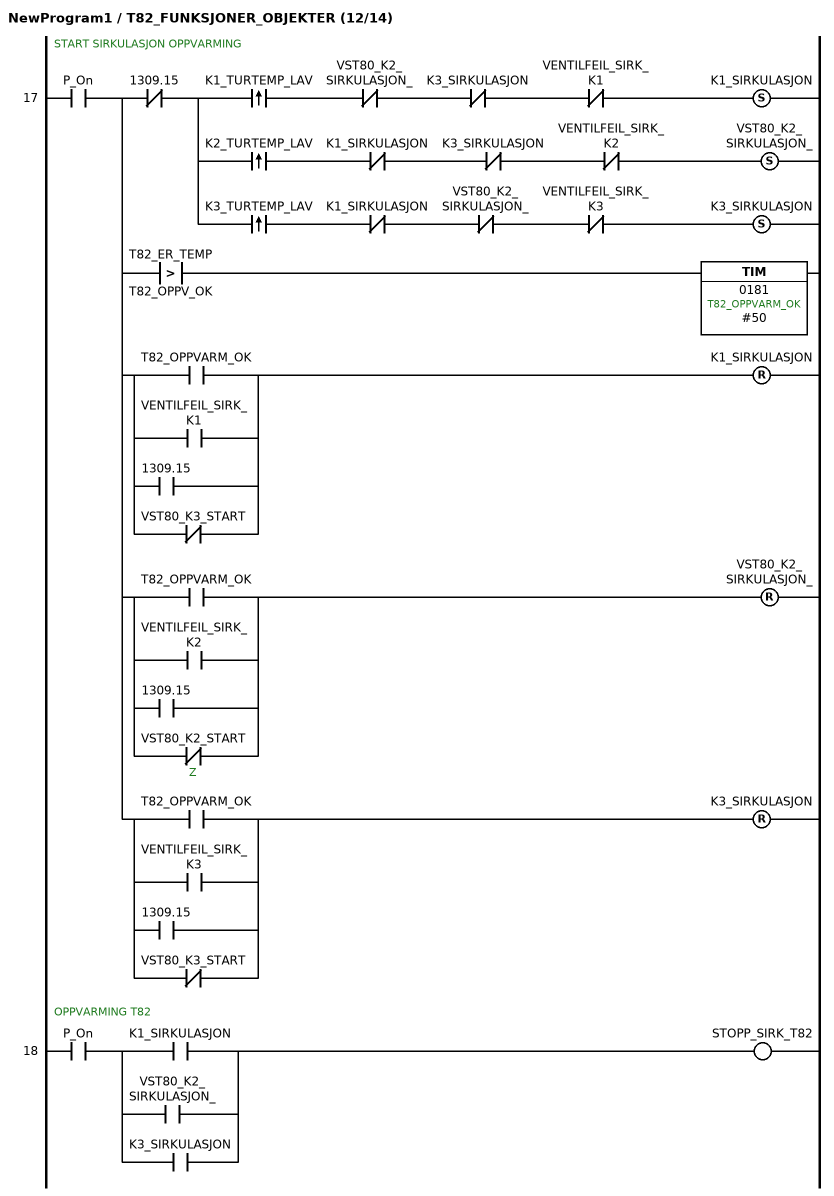
; rung 17: START SIRKULASJON OPPVARMING
LD P_On
OUT TR0
ANDNOT 1309.15
OUT TR1
@AND K1_TURTEMP_LAV
ANDNOT VST80_K2_SIRKULASJON_
ANDNOT K3_SIRKULASJON
ANDNOT VENTILFEIL_SIRK_K1
SET K1_SIRKULASJON
LD TR1
@AND K2_TURTEMP_LAV
ANDNOT K1_SIRKULASJON
ANDNOT K3_SIRKULASJON
ANDNOT VENTILFEIL_SIRK_K2
SET VST80_K2_SIRKULASJON_
LD TR1
@AND K3_TURTEMP_LAV
ANDNOT K1_SIRKULASJON
ANDNOT VST80_K2_SIRKULASJON_
ANDNOT VENTILFEIL_SIRK_K3
SET K3_SIRKULASJON
LD TR0
AND>(320) T82_ER_TEMP T82_OPPV_OK
TIM 0181 #50  ; T82_OPPVARM_OK
LD TR0
LD T82_OPPVARM_OK
OR VENTILFEIL_SIRK_K1
OR 1309.15
ORNOT VST80_K3_START
ANDLD
RSET K1_SIRKULASJON
LD TR0
LD T82_OPPVARM_OK
OR VENTILFEIL_SIRK_K2
OR 1309.15
ORNOT VST80_K2_START  ; Z
ANDLD
RSET VST80_K2_SIRKULASJON_
LD TR0
LD T82_OPPVARM_OK
OR VENTILFEIL_SIRK_K3
OR 1309.15
ORNOT VST80_K3_START
ANDLD
RSET K3_SIRKULASJON
; rung 18: OPPVARMING T82
LD P_On
LD K1_SIRKULASJON
OR VST80_K2_SIRKULASJON_
OR K3_SIRKULASJON
ANDLD
OUT STOPP_SIRK_T82

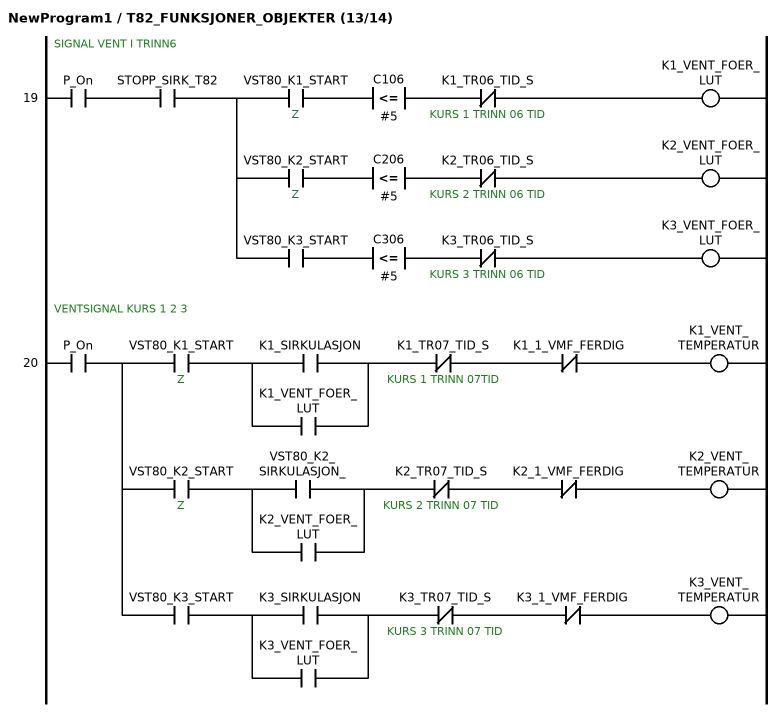
; rung 19: SIGNAL VENT I TRINN6
LD P_On
AND STOPP_SIRK_T82
OUT TR0
AND VST80_K1_START  ; Z
AND<=(315) C106 #5
ANDNOT K1_TR06_TID_S  ; KURS 1 TRINN 06 TID
OUT K1_VENT_FOER_LUT
LD TR0
AND VST80_K2_START  ; Z
AND<=(315) C206 #5
ANDNOT K2_TR06_TID_S  ; KURS 2 TRINN 06 TID
OUT K2_VENT_FOER_LUT
LD TR0
AND VST80_K3_START
AND<=(315) C306 #5
ANDNOT K3_TR06_TID_S  ; KURS 3 TRINN 06 TID
OUT K3_VENT_FOER_LUT
; rung 20: VENTSIGNAL KURS 1 2 3
LD P_On
OUT TR0
AND VST80_K1_START  ; Z
LD K1_SIRKULASJON
OR K1_VENT_FOER_LUT
ANDLD
ANDNOT K1_TR07_TID_S  ; KURS 1 TRINN 07TID
ANDNOT K1_1_VMF_FERDIG
OUT K1_VENT_TEMPERATUR
LD TR0
AND VST80_K2_START  ; Z
LD VST80_K2_SIRKULASJON_
OR K2_VENT_FOER_LUT
ANDLD
ANDNOT K2_TR07_TID_S  ; KURS 2 TRINN 07 TID
ANDNOT K2_1_VMF_FERDIG
OUT K2_VENT_TEMPERATUR
LD TR0
AND VST80_K3_START
LD K3_SIRKULASJON
OR K3_VENT_FOER_LUT
ANDLD
ANDNOT K3_TR07_TID_S  ; KURS 3 TRINN 07 TID
ANDNOT K3_1_VMF_FERDIG
OUT K3_VENT_TEMPERATUR

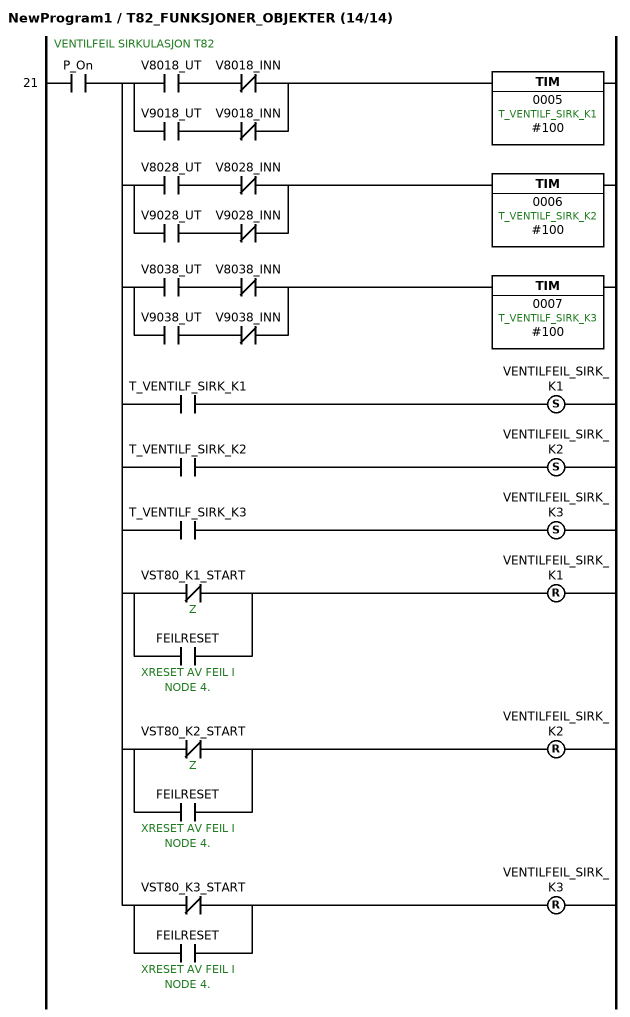
; rung 21: VENTILFEIL SIRKULASJON T82
LD P_On
OUT TR0
LD V8018_UT
ANDNOT V8018_INN
LD V9018_UT
ANDNOT V9018_INN
ORLD
ANDLD
TIM 0005 #100  ; T_VENTILF_SIRK_K1
LD TR0
LD V8028_UT
ANDNOT V8028_INN
LD V9028_UT
ANDNOT V9028_INN
ORLD
ANDLD
TIM 0006 #100  ; T_VENTILF_SIRK_K2
LD TR0
LD V8038_UT
ANDNOT V8038_INN
LD V9038_UT
ANDNOT V9038_INN
ORLD
ANDLD
TIM 0007 #100  ; T_VENTILF_SIRK_K3
LD TR0
AND T_VENTILF_SIRK_K1
SET VENTILFEIL_SIRK_K1
LD TR0
AND T_VENTILF_SIRK_K2
SET VENTILFEIL_SIRK_K2
LD TR0
AND T_VENTILF_SIRK_K3
SET VENTILFEIL_SIRK_K3
LD TR0
LDNOT VST80_K1_START  ; Z
OR FEILRESET  ; XRESET AV FEIL I NODE 4.
ANDLD
RSET VENTILFEIL_SIRK_K1
LD TR0
LDNOT VST80_K2_START  ; Z
OR FEILRESET  ; XRESET AV FEIL I NODE 4.
ANDLD
RSET VENTILFEIL_SIRK_K2
LD TR0
LDNOT VST80_K3_START
OR FEILRESET  ; XRESET AV FEIL I NODE 4.
ANDLD
RSET VENTILFEIL_SIRK_K3
; rung 22: Ingen_kommentar_funnet

### Section T83_NIVÅ_TEMP_KONDUKTIVITET

